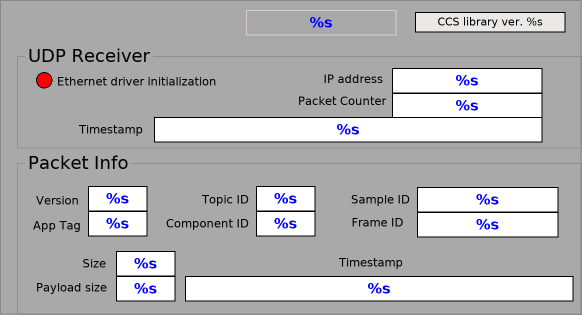
VISUALIZATION GUI_TEMPLATE_MUDPI_RECEIVER  // 582x315
VAR_INPUT
	m_DeviceName : STRING;
END_VAR
VAR_IN_OUT
	m_Instance : FB_MUDPI_RECEIVER;
END_VAR
    GroupBox (17,48 565x100), "UDP Receiver"
        Rectangle (375,20 150x25), "%s", text variable: m_Instance.udp_info.ipv4Adr
            OnMouseDown: write the text variable via Edit
        Label (285,18 84x26), "IP address"
        Label (37,19 240x29), "Ethernet driver initialization"
        Ellipse (19,24 16x16), tooltip "RED - False GREEN - True", colour toggle: m_Instance.udp_info.bDriverInitialization
        Label (265,40 107x26), "Packet Counter"
        Rectangle (375,45 150x25), "%s", text variable: m_Instance.udp_info.nReceivedPackets
            OnMouseDown: write the text variable via Edit
        Rectangle (137,69 388x25), "%s", tooltip "Time used for Simulation. Press "Copy UTC" or "Copy Local" button to get the time in correct format and then modify it for your needs.", text variable: m_Instance.udp_info.sNotification
            OnMouseDown: write the text variable via Default
        Label (56,70 76x23), "Timestamp"
    Rectangle (246,10 150x25), "%s", text variable: m_Instance.instance_name
    Rectangle (415,12 150x20), "CCS library ver. %s", text variable: m_Instance.sLibVersion
    GroupBox (17,155 565x160), "Packet Info"
        Rectangle (71,31 59x25), "%s", text variable: m_Instance.packet_info.version
            OnMouseDown: write the text variable via Edit
        Rectangle (71,56 59x25), "%s", text variable: m_Instance.packet_info.appTag
            OnMouseDown: write the text variable via Edit
        Label (6,31 59x29), "Version"
        Label (6,56 61x29), "App Tag"
        Label (329,30 67x29), "Sample ID"
        Rectangle (400,32 141x25), "%s", text variable: m_Instance.packet_info.sampleId
            OnMouseDown: write the text variable via Edit
        Rectangle (239,31 59x25), "%s", text variable: m_Instance.packet_info.topicId
            OnMouseDown: write the text variable via Edit
        Label (176,30 59x29), "Topic ID"
        Label (148,54 87x29), "Component ID"
        Rectangle (239,56 59x25), "%s", text variable: m_Instance.packet_info.componentId
            OnMouseDown: write the text variable via Edit
        Rectangle (400,57 141x25), "%s", text variable: m_Instance.packet_info.frameId
            OnMouseDown: write the text variable via Edit
        Label (304,53 89x29), "Frame ID"
        Label (316,96 76x23), "Timestamp"
        Rectangle (168,121 388x25), "%s", tooltip "Time used for Simulation. Press "Copy UTC" or "Copy Local" button to get the time in correct format and then modify it for your needs.", text variable: m_Instance.packet_info.timestamp
            OnMouseDown: write the text variable via Default
        Label (25,94 67x29), "Size"
        Label (12,118 81x29), "Payload size"
        Rectangle (99,96 59x25), "%s", text variable: m_Instance.packet_info.size
            OnMouseDown: write the text variable via Edit
        Rectangle (99,121 59x25), "%s", text variable: m_Instance.packet_info.payloadSize
            OnMouseDown: write the text variable via Edit
END_VISUALIZATION

(* stored: Version 1.1.0.1, ProductVersion 3.1.4024.11
   Visu GUI_TEMPLATE_MUDPI_RECEIVER: Id {9265c798-38b0-452a-bfbb-7e96b4d7ae66} *)
